INTERFACE ITF_1_Robot EXTENDS ITF_0_BaseComponent

METHOD EnableRobot : BOOL
VAR_INPUT
END_VAR
END_METHOD

METHOD DisableRobot : BOOL
VAR_INPUT
END_VAR
END_METHOD

METHOD ResetRobot : BOOL
VAR_INPUT
END_VAR
END_METHOD

METHOD Stop : BOOL
VAR_INPUT
END_VAR
END_METHOD

METHOD Pause : BOOL
VAR_INPUT
END_VAR
END_METHOD

METHOD Resume : BOOL
VAR_INPUT
END_VAR
END_METHOD

METHOD SetOperationMode : BOOL
VAR_INPUT
    mode : eMode;
END_VAR
END_METHOD

METHOD SetSpeedOverride : BOOL
VAR_INPUT
    factor : LREAL;
END_VAR
END_METHOD

PROPERTY CommunicationReady : BOOL
GET
END_GET
SET
END_SET
END_PROPERTY

PROPERTY RobotEnabled : BOOL
GET
END_GET
SET
END_SET
END_PROPERTY

PROPERTY RobotReady : BOOL
GET
END_GET
SET
END_SET
END_PROPERTY

PROPERTY Busy : BOOL
GET
END_GET
SET
END_SET
END_PROPERTY

PROPERTY RobotMoving : BOOL
GET
END_GET
SET
END_SET
END_PROPERTY

PROPERTY RobotError : BOOL
GET
END_GET
END_PROPERTY

PROPERTY Mode : eMode
GET
END_GET
SET
END_SET
END_PROPERTY

PROPERTY Collision : BOOL
GET
END_GET
END_PROPERTY

END_INTERFACE

(* stored: Version 1.1.0.1, ProductVersion 3.1.4026.18
   Itf ITF_1_Robot: Id {a6d29cf6-e144-4e1d-bf83-e7b2be10a693}
   Method EnableRobot: Id {0f3f76ce-0c24-431f-b0cb-d24dc0415a91}
   Method DisableRobot: Id {1f5c5c05-2dcb-40b6-85b7-e14de76733ca}
   Method ResetRobot: Id {6bd7f640-7106-49dd-a5cd-96054e8ed6ff}
   Method Stop: Id {1643e2ed-a195-4fb9-bcc2-d0e7b52e61fb}
   Method Pause: Id {a219643f-8e25-47f8-b4f4-e2335d3e6ead}
   Method Resume: Id {bd189bc6-367b-4937-84f7-9d3aaa9bc52d}
   Method SetOperationMode: Id {4a5f6fe2-c0ac-4a0a-ac11-a7823ebd0b5f}
   Method SetSpeedOverride: Id {a5c3a683-3c13-4a4d-9450-cd749be2641d}
   Property CommunicationReady: Id {0f7c4d71-4dca-482c-958c-60b22ceffb31}
   Get Get: Id {ec70d493-1735-4eee-8f28-8fedbca6eeaa}
   Set Set: Id {f8dbcf8c-d3f0-41e0-b458-f68b9e03f4ec}
   Property RobotEnabled: Id {95536b20-47f3-4d85-8846-0f4cc34c4b04}
   Get Get: Id {3c40598d-bbaa-48a0-aee9-84c6b65300d9}
   Set Set: Id {f92a9311-3db4-4205-a650-2523b8b0dc13}
   Property RobotReady: Id {32f7ce06-a917-40aa-a63a-9d645daf1000}
   Get Get: Id {78af0e9a-e888-424b-9875-3b938dfeb7c8}
   Set Set: Id {bb3142fc-b931-4e52-8d9e-2089283ba332}
   Property Busy: Id {40247604-64eb-4bf8-bd71-13681de4b94c}
   Get Get: Id {4e01a15e-27d1-4a27-8b69-b9e60512da87}
   Set Set: Id {d80c3a91-9c5e-4e41-9c00-52957c4ee123}
   Property RobotMoving: Id {3ed4e89d-1bdc-4ba3-aaab-47d06e86a2de}
   Get Get: Id {1fbb8003-a640-4c09-a91d-be28a7a884bd}
   Set Set: Id {a33a2cc5-228b-4b66-98ef-d7a791374683}
   Property RobotError: Id {3513c5a9-7727-46e6-a0de-4cd54a023352}
   Get Get: Id {ae41d1b9-6a22-46bc-9839-e1e32660158a}
   Property Mode: Id {884c7276-7307-49dc-816b-0ffea2c4cba8}
   Get Get: Id {b3dfabc4-c456-4561-bf20-1871e1ecd3cb}
   Set Set: Id {d0624bcc-9094-492f-8b17-2c7b6b805814}
   Property Collision: Id {ca6d4356-07c4-4425-9b71-7b2c8a3d9b7b}
   Get Get: Id {e72de0d8-8a39-42e4-884d-411c14a93e5c} *)
